FUNCTION_BLOCK FB_EL922x_ChannelBasic_1 IMPLEMENTS ITF_EL922x_ChannelBasic
VAR_INPUT
END_VAR
VAR_OUTPUT
END_VAR
VAR
	_Chn : EL922x_ChannelBasic;
END_VAR

END_FUNCTION_BLOCK

(* stored: Version 1.1.0.1, ProductVersion 3.1.4024.5
   POU FB_EL922x_ChannelBasic_1: Id {217eb7e0-aa40-4892-a9c6-20fefeef290a}, SpecialFunc None *)
